{attribute 'GeneratedUsingTerminal: AX8108-0100-0101-0101'}
{attribute addProperty BoxType "AX8108-0100-0101-0101"}
{attribute addProperty Id "FSOEAT %I*FSOE_13BCEA3F2"}
{attribute addProperty CRC "3443497619"}
{attribute addProperty Size "2"}
TYPE FSLOGIC_Inputs_CD3F9A93 :
STRUCT
	{attribute addProperty Name "FSOE"}
	FSOE AT %I* : FSOE_13BCEA3F;
END_STRUCT
END_TYPE

(* stored: Version 1.2.0.0, ProductVersion 3.1.4024.9
   DUT FSLOGIC_Inputs_CD3F9A93: Id {e7f08109-1433-4810-a1b3-9ee23304d591} *)
